SUBAPPLICATION Uebung_011g1_AX (* Numeric Value Input -- multiple IOObservers *)
  (* Standard: 61499-2; Description: Copyright (c) 2023 Meisterschulen am Ostbahnhof This program and the accompanying materials are made available under the terms of the Eclipse Public License 2.0 which is available at https://www.eclipse.org/legal/epl-2.0/ SPDX-License-Identifier: EPL-2.0 *)
  (* Version 1.1, 2026-05-05, Franz Höpfinger, Meisterschulen am Ostbahnhof, multiple IOObservers *)
  (* Version 1.0, 2023-10-23, Franz Höpfinger, Meisterschulen am Ostbahnhof, initial API and implementation and/or initial documentation *)
  PACKAGE Uebungen;
  IMPORT Uebungen::const::UT::DefaultPool::InputNumber_I1;
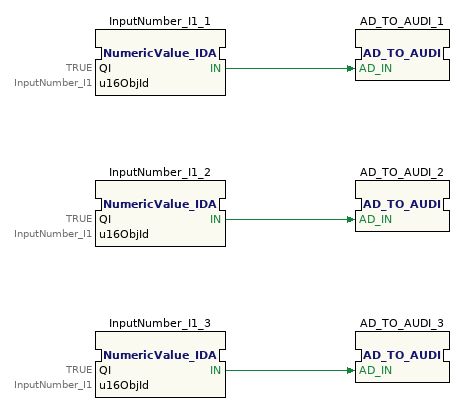
  FBS
    InputNumber_I1_1 : isobus::UT::io::NumericValue::NumericValue_IDA(QI := TRUE, u16ObjId := InputNumber_I1);
    InputNumber_I1_2 : isobus::UT::io::NumericValue::NumericValue_IDA(QI := TRUE, u16ObjId := InputNumber_I1);
    InputNumber_I1_3 : isobus::UT::io::NumericValue::NumericValue_IDA(QI := TRUE, u16ObjId := InputNumber_I1);
    AD_TO_AUDI_1 : adapter::conversion::unidirectional::AD_TO_AUDI;
    AD_TO_AUDI_2 : adapter::conversion::unidirectional::AD_TO_AUDI;
    AD_TO_AUDI_3 : adapter::conversion::unidirectional::AD_TO_AUDI;
  END_FBS
  ADAPTER_CONNECTIONS
    InputNumber_I1_1.IN TO AD_TO_AUDI_1.AD_IN;
    InputNumber_I1_2.IN TO AD_TO_AUDI_2.AD_IN;
    InputNumber_I1_3.IN TO AD_TO_AUDI_3.AD_IN;
  END_CONNECTIONS
END_SUBAPPLICATION
